// TIA Portal V17 export
// export: Created 2024-08-21T14:00:35.6590346Z, ExportSetting WithDefaults, DisplayName Totally Integrated Automation Portal, DisplayVersion V17 Update 4, DisplayName TIA Portal Openness, DisplayVersion V17 Update 4, DisplayName TIA Portal Version Control Interface, DisplayVersion V17, DisplayName STEP 7 Professional, DisplayVersion V17 Update 4, DisplayName STEP 7 Safety, DisplayVersion V17, DisplayName WinCC Advanced, DisplayVersion V17 Update 4
FUNCTION "IO" : Void   // FC1, LAD
{ S7_Optimized_Access := 'TRUE' }
VERSION : 0.1
// stored: AutoNumber false, IsIECCheckEnabled false, SetENOAutomatically false, UDAEnableTagReadback false
BEGIN

REGION Network 1: Status e alarme elevatória principal 1
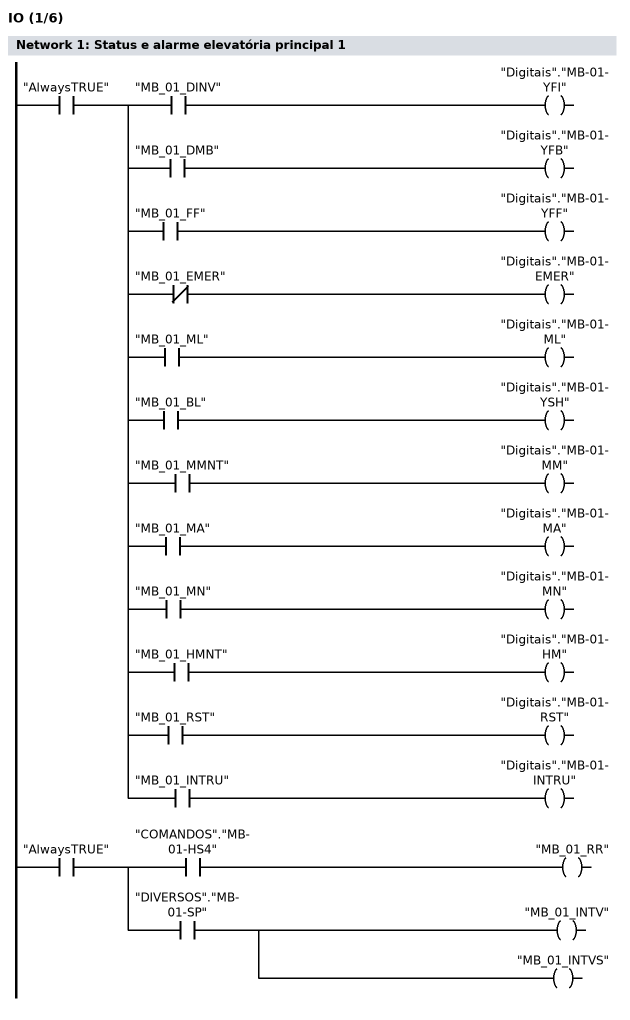
   RUNG wire#powerrail
      Contact( "AlwaysTRUE" )
      wire#w1
      Contact( "MB_01_DINV" )
      Coil( "Digitais"."MB-01-YFI" )
   END_RUNG
   RUNG wire#w1
      Contact( "MB_01_DMB" )
      Coil( "Digitais"."MB-01-YFB" )
   END_RUNG
   RUNG wire#w1
      Contact( "MB_01_FF" )
      Coil( "Digitais"."MB-01-YFF" )
   END_RUNG
   RUNG wire#w1
      I_Contact( "MB_01_EMER" )
      Coil( "Digitais"."MB-01-EMER" )
   END_RUNG
   RUNG wire#w1
      Contact( "MB_01_ML" )
      Coil( "Digitais"."MB-01-ML" )
   END_RUNG
   RUNG wire#w1
      Contact( "MB_01_BL" )
      Coil( "Digitais"."MB-01-YSH" )
   END_RUNG
   RUNG wire#w1
      Contact( "MB_01_MMNT" )
      Coil( "Digitais"."MB-01-MM" )
   END_RUNG
   RUNG wire#w1
      Contact( "MB_01_MA" )
      Coil( "Digitais"."MB-01-MA" )
   END_RUNG
   RUNG wire#w1
      Contact( "MB_01_MN" )
      Coil( "Digitais"."MB-01-MN" )
   END_RUNG
   RUNG wire#w1
      Contact( "MB_01_HMNT" )
      Coil( "Digitais"."MB-01-HM" )
   END_RUNG
   RUNG wire#w1
      Contact( "MB_01_RST" )
      Coil( "Digitais"."MB-01-RST" )
   END_RUNG
   RUNG wire#w1
      Contact( "MB_01_INTRU" )
      Coil( "Digitais"."MB-01-INTRU" )
   END_RUNG
   RUNG wire#powerrail
      Contact( "AlwaysTRUE" )
      wire#w2
      Contact( "COMANDOS"."MB-01-HS4" )
      Coil( "MB_01_RR" )
   END_RUNG
   RUNG wire#w2
      Contact( "DIVERSOS"."MB-01-SP" )
      wire#w3
      Coil( "MB_01_INTV" )
   END_RUNG
   RUNG wire#w3
      Coil( "MB_01_INTVS" )
   END_RUNG
   // the same network as SCL:
   "Digitais"."MB-01-YFI" := "AlwaysTRUE" AND "MB_01_DINV";
   "Digitais"."MB-01-YFB" := "AlwaysTRUE" AND "MB_01_DMB";
   "Digitais"."MB-01-YFF" := "AlwaysTRUE" AND "MB_01_FF";
   "Digitais"."MB-01-EMER" := "AlwaysTRUE" AND NOT "MB_01_EMER";
   "Digitais"."MB-01-ML" := "AlwaysTRUE" AND "MB_01_ML";
   "Digitais"."MB-01-YSH" := "AlwaysTRUE" AND "MB_01_BL";
   "Digitais"."MB-01-MM" := "AlwaysTRUE" AND "MB_01_MMNT";
   "Digitais"."MB-01-MA" := "AlwaysTRUE" AND "MB_01_MA";
   "Digitais"."MB-01-MN" := "AlwaysTRUE" AND "MB_01_MN";
   "Digitais"."MB-01-HM" := "AlwaysTRUE" AND "MB_01_HMNT";
   "Digitais"."MB-01-RST" := "AlwaysTRUE" AND "MB_01_RST";
   "Digitais"."MB-01-INTRU" := "AlwaysTRUE" AND "MB_01_INTRU";
   "MB_01_RR" := "AlwaysTRUE" AND "COMANDOS"."MB-01-HS4";
   "MB_01_INTV" := "AlwaysTRUE" AND "DIVERSOS"."MB-01-SP";
   "MB_01_INTVS" := "MB_01_INTV";
END_REGION

REGION Network 2: Status e alarme elevatória principal 2
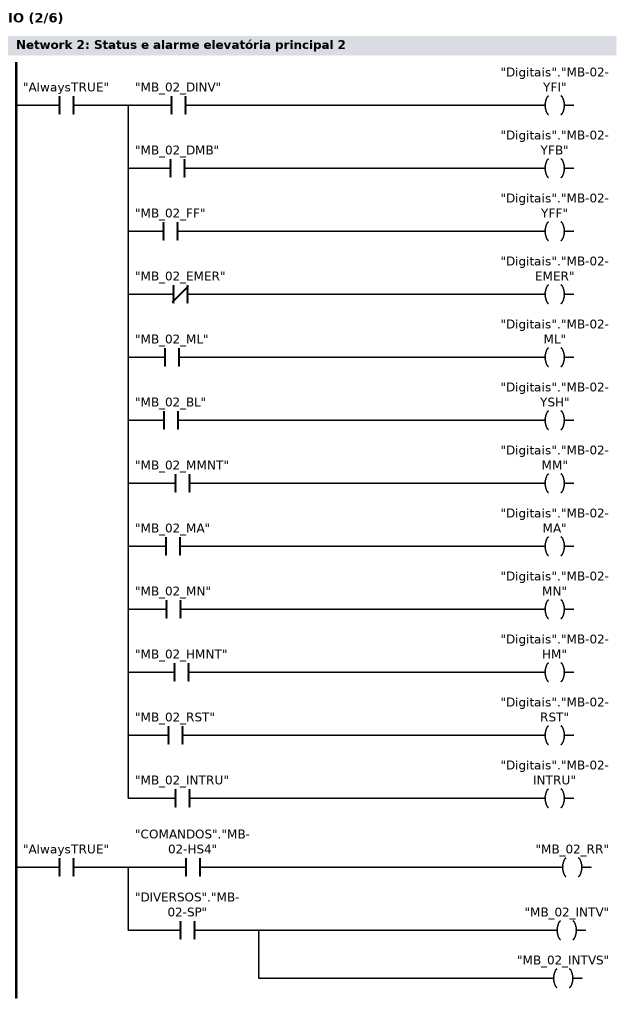
   RUNG wire#powerrail
      Contact( "AlwaysTRUE" )
      wire#w1
      Contact( "MB_02_DINV" )
      Coil( "Digitais"."MB-02-YFI" )
   END_RUNG
   RUNG wire#w1
      Contact( "MB_02_DMB" )
      Coil( "Digitais"."MB-02-YFB" )
   END_RUNG
   RUNG wire#w1
      Contact( "MB_02_FF" )
      Coil( "Digitais"."MB-02-YFF" )
   END_RUNG
   RUNG wire#w1
      I_Contact( "MB_02_EMER" )
      Coil( "Digitais"."MB-02-EMER" )
   END_RUNG
   RUNG wire#w1
      Contact( "MB_02_ML" )
      Coil( "Digitais"."MB-02-ML" )
   END_RUNG
   RUNG wire#w1
      Contact( "MB_02_BL" )
      Coil( "Digitais"."MB-02-YSH" )
   END_RUNG
   RUNG wire#w1
      Contact( "MB_02_MMNT" )
      Coil( "Digitais"."MB-02-MM" )
   END_RUNG
   RUNG wire#w1
      Contact( "MB_02_MA" )
      Coil( "Digitais"."MB-02-MA" )
   END_RUNG
   RUNG wire#w1
      Contact( "MB_02_MN" )
      Coil( "Digitais"."MB-02-MN" )
   END_RUNG
   RUNG wire#w1
      Contact( "MB_02_HMNT" )
      Coil( "Digitais"."MB-02-HM" )
   END_RUNG
   RUNG wire#w1
      Contact( "MB_02_RST" )
      Coil( "Digitais"."MB-02-RST" )
   END_RUNG
   RUNG wire#w1
      Contact( "MB_02_INTRU" )
      Coil( "Digitais"."MB-02-INTRU" )
   END_RUNG
   RUNG wire#powerrail
      Contact( "AlwaysTRUE" )
      wire#w2
      Contact( "COMANDOS"."MB-02-HS4" )
      Coil( "MB_02_RR" )
   END_RUNG
   RUNG wire#w2
      Contact( "DIVERSOS"."MB-02-SP" )
      wire#w3
      Coil( "MB_02_INTV" )
   END_RUNG
   RUNG wire#w3
      Coil( "MB_02_INTVS" )
   END_RUNG
   // the same network as SCL:
   "Digitais"."MB-02-YFI" := "AlwaysTRUE" AND "MB_02_DINV";
   "Digitais"."MB-02-YFB" := "AlwaysTRUE" AND "MB_02_DMB";
   "Digitais"."MB-02-YFF" := "AlwaysTRUE" AND "MB_02_FF";
   "Digitais"."MB-02-EMER" := "AlwaysTRUE" AND NOT "MB_02_EMER";
   "Digitais"."MB-02-ML" := "AlwaysTRUE" AND "MB_02_ML";
   "Digitais"."MB-02-YSH" := "AlwaysTRUE" AND "MB_02_BL";
   "Digitais"."MB-02-MM" := "AlwaysTRUE" AND "MB_02_MMNT";
   "Digitais"."MB-02-MA" := "AlwaysTRUE" AND "MB_02_MA";
   "Digitais"."MB-02-MN" := "AlwaysTRUE" AND "MB_02_MN";
   "Digitais"."MB-02-HM" := "AlwaysTRUE" AND "MB_02_HMNT";
   "Digitais"."MB-02-RST" := "AlwaysTRUE" AND "MB_02_RST";
   "Digitais"."MB-02-INTRU" := "AlwaysTRUE" AND "MB_02_INTRU";
   "MB_02_RR" := "AlwaysTRUE" AND "COMANDOS"."MB-02-HS4";
   "MB_02_INTV" := "AlwaysTRUE" AND "DIVERSOS"."MB-02-SP";
   "MB_02_INTVS" := "MB_02_INTV";
END_REGION

REGION Network 3: Status e alarme elevatória principal 3
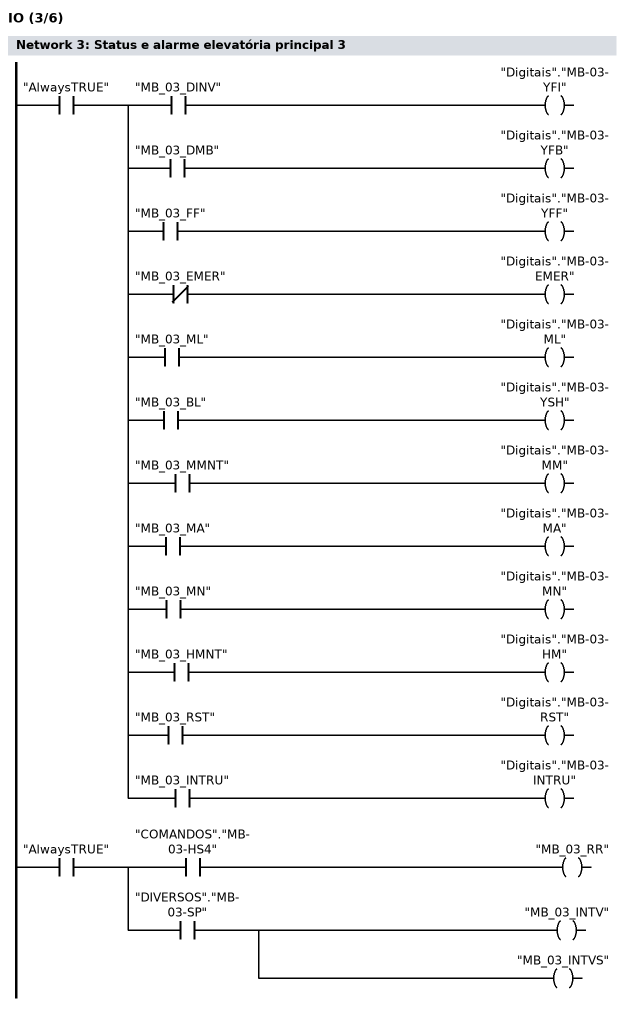
   RUNG wire#powerrail
      Contact( "AlwaysTRUE" )
      wire#w1
      Contact( "MB_03_DINV" )
      Coil( "Digitais"."MB-03-YFI" )
   END_RUNG
   RUNG wire#w1
      Contact( "MB_03_DMB" )
      Coil( "Digitais"."MB-03-YFB" )
   END_RUNG
   RUNG wire#w1
      Contact( "MB_03_FF" )
      Coil( "Digitais"."MB-03-YFF" )
   END_RUNG
   RUNG wire#w1
      I_Contact( "MB_03_EMER" )
      Coil( "Digitais"."MB-03-EMER" )
   END_RUNG
   RUNG wire#w1
      Contact( "MB_03_ML" )
      Coil( "Digitais"."MB-03-ML" )
   END_RUNG
   RUNG wire#w1
      Contact( "MB_03_BL" )
      Coil( "Digitais"."MB-03-YSH" )
   END_RUNG
   RUNG wire#w1
      Contact( "MB_03_MMNT" )
      Coil( "Digitais"."MB-03-MM" )
   END_RUNG
   RUNG wire#w1
      Contact( "MB_03_MA" )
      Coil( "Digitais"."MB-03-MA" )
   END_RUNG
   RUNG wire#w1
      Contact( "MB_03_MN" )
      Coil( "Digitais"."MB-03-MN" )
   END_RUNG
   RUNG wire#w1
      Contact( "MB_03_HMNT" )
      Coil( "Digitais"."MB-03-HM" )
   END_RUNG
   RUNG wire#w1
      Contact( "MB_03_RST" )
      Coil( "Digitais"."MB-03-RST" )
   END_RUNG
   RUNG wire#w1
      Contact( "MB_03_INTRU" )
      Coil( "Digitais"."MB-03-INTRU" )
   END_RUNG
   RUNG wire#powerrail
      Contact( "AlwaysTRUE" )
      wire#w2
      Contact( "COMANDOS"."MB-03-HS4" )
      Coil( "MB_03_RR" )
   END_RUNG
   RUNG wire#w2
      Contact( "DIVERSOS"."MB-03-SP" )
      wire#w3
      Coil( "MB_03_INTV" )
   END_RUNG
   RUNG wire#w3
      Coil( "MB_03_INTVS" )
   END_RUNG
   // the same network as SCL:
   "Digitais"."MB-03-YFI" := "AlwaysTRUE" AND "MB_03_DINV";
   "Digitais"."MB-03-YFB" := "AlwaysTRUE" AND "MB_03_DMB";
   "Digitais"."MB-03-YFF" := "AlwaysTRUE" AND "MB_03_FF";
   "Digitais"."MB-03-EMER" := "AlwaysTRUE" AND NOT "MB_03_EMER";
   "Digitais"."MB-03-ML" := "AlwaysTRUE" AND "MB_03_ML";
   "Digitais"."MB-03-YSH" := "AlwaysTRUE" AND "MB_03_BL";
   "Digitais"."MB-03-MM" := "AlwaysTRUE" AND "MB_03_MMNT";
   "Digitais"."MB-03-MA" := "AlwaysTRUE" AND "MB_03_MA";
   "Digitais"."MB-03-MN" := "AlwaysTRUE" AND "MB_03_MN";
   "Digitais"."MB-03-HM" := "AlwaysTRUE" AND "MB_03_HMNT";
   "Digitais"."MB-03-RST" := "AlwaysTRUE" AND "MB_03_RST";
   "Digitais"."MB-03-INTRU" := "AlwaysTRUE" AND "MB_03_INTRU";
   "MB_03_RR" := "AlwaysTRUE" AND "COMANDOS"."MB-03-HS4";
   "MB_03_INTV" := "AlwaysTRUE" AND "DIVERSOS"."MB-03-SP";
   "MB_03_INTVS" := "MB_03_INTV";
END_REGION

REGION Network 4: Status e alarme elevatória principal 4
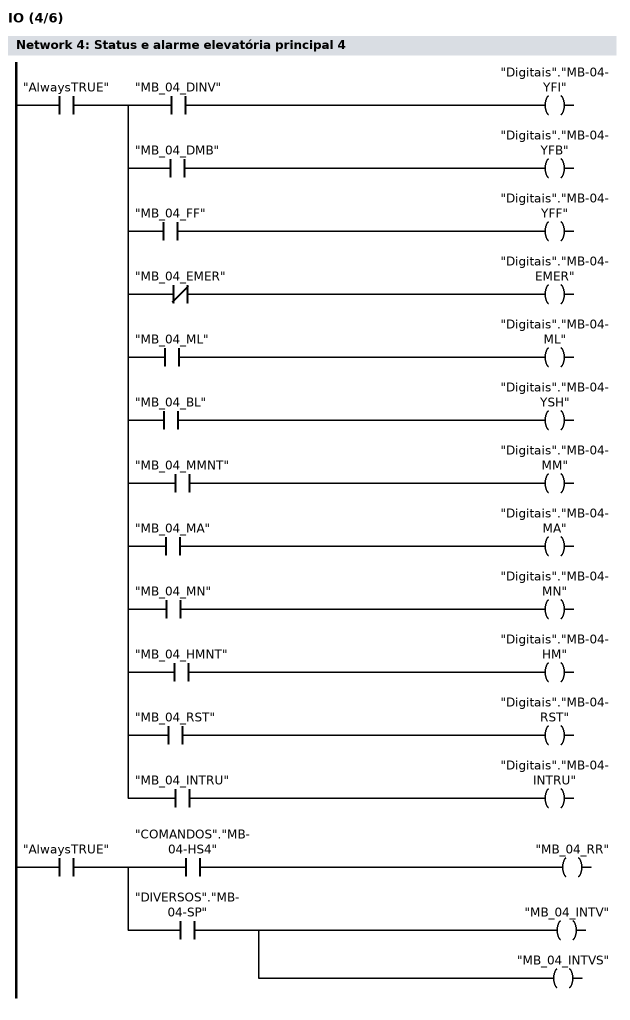
   RUNG wire#powerrail
      Contact( "AlwaysTRUE" )
      wire#w1
      Contact( "MB_04_DINV" )
      Coil( "Digitais"."MB-04-YFI" )
   END_RUNG
   RUNG wire#w1
      Contact( "MB_04_DMB" )
      Coil( "Digitais"."MB-04-YFB" )
   END_RUNG
   RUNG wire#w1
      Contact( "MB_04_FF" )
      Coil( "Digitais"."MB-04-YFF" )
   END_RUNG
   RUNG wire#w1
      I_Contact( "MB_04_EMER" )
      Coil( "Digitais"."MB-04-EMER" )
   END_RUNG
   RUNG wire#w1
      Contact( "MB_04_ML" )
      Coil( "Digitais"."MB-04-ML" )
   END_RUNG
   RUNG wire#w1
      Contact( "MB_04_BL" )
      Coil( "Digitais"."MB-04-YSH" )
   END_RUNG
   RUNG wire#w1
      Contact( "MB_04_MMNT" )
      Coil( "Digitais"."MB-04-MM" )
   END_RUNG
   RUNG wire#w1
      Contact( "MB_04_MA" )
      Coil( "Digitais"."MB-04-MA" )
   END_RUNG
   RUNG wire#w1
      Contact( "MB_04_MN" )
      Coil( "Digitais"."MB-04-MN" )
   END_RUNG
   RUNG wire#w1
      Contact( "MB_04_HMNT" )
      Coil( "Digitais"."MB-04-HM" )
   END_RUNG
   RUNG wire#w1
      Contact( "MB_04_RST" )
      Coil( "Digitais"."MB-04-RST" )
   END_RUNG
   RUNG wire#w1
      Contact( "MB_04_INTRU" )
      Coil( "Digitais"."MB-04-INTRU" )
   END_RUNG
   RUNG wire#powerrail
      Contact( "AlwaysTRUE" )
      wire#w2
      Contact( "COMANDOS"."MB-04-HS4" )
      Coil( "MB_04_RR" )
   END_RUNG
   RUNG wire#w2
      Contact( "DIVERSOS"."MB-04-SP" )
      wire#w3
      Coil( "MB_04_INTV" )
   END_RUNG
   RUNG wire#w3
      Coil( "MB_04_INTVS" )
   END_RUNG
   // the same network as SCL:
   "Digitais"."MB-04-YFI" := "AlwaysTRUE" AND "MB_04_DINV";
   "Digitais"."MB-04-YFB" := "AlwaysTRUE" AND "MB_04_DMB";
   "Digitais"."MB-04-YFF" := "AlwaysTRUE" AND "MB_04_FF";
   "Digitais"."MB-04-EMER" := "AlwaysTRUE" AND NOT "MB_04_EMER";
   "Digitais"."MB-04-ML" := "AlwaysTRUE" AND "MB_04_ML";
   "Digitais"."MB-04-YSH" := "AlwaysTRUE" AND "MB_04_BL";
   "Digitais"."MB-04-MM" := "AlwaysTRUE" AND "MB_04_MMNT";
   "Digitais"."MB-04-MA" := "AlwaysTRUE" AND "MB_04_MA";
   "Digitais"."MB-04-MN" := "AlwaysTRUE" AND "MB_04_MN";
   "Digitais"."MB-04-HM" := "AlwaysTRUE" AND "MB_04_HMNT";
   "Digitais"."MB-04-RST" := "AlwaysTRUE" AND "MB_04_RST";
   "Digitais"."MB-04-INTRU" := "AlwaysTRUE" AND "MB_04_INTRU";
   "MB_04_RR" := "AlwaysTRUE" AND "COMANDOS"."MB-04-HS4";
   "MB_04_INTV" := "AlwaysTRUE" AND "DIVERSOS"."MB-04-SP";
   "MB_04_INTVS" := "MB_04_INTV";
END_REGION

REGION Network 5: Status e alarme PCM-E-CF-01-04
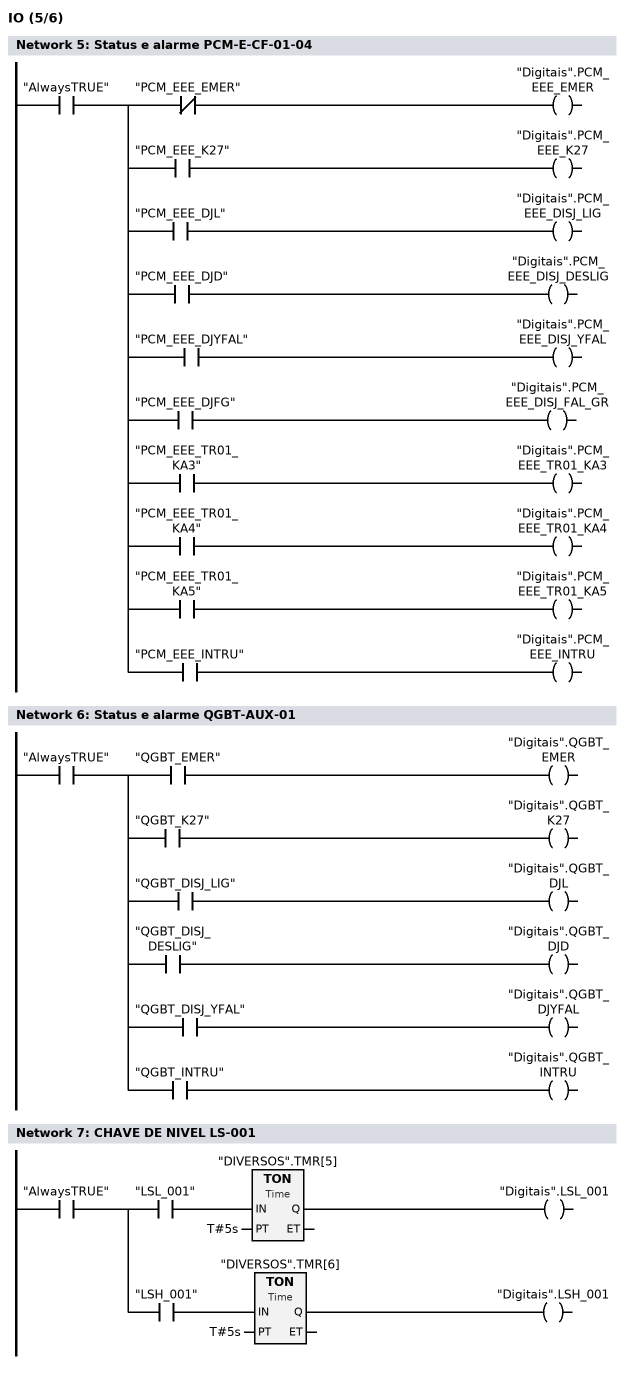
   RUNG wire#powerrail
      Contact( "AlwaysTRUE" )
      wire#w1
      I_Contact( "PCM_EEE_EMER" )
      Coil( "Digitais".PCM_EEE_EMER )
   END_RUNG
   RUNG wire#w1
      Contact( "PCM_EEE_K27" )
      Coil( "Digitais".PCM_EEE_K27 )
   END_RUNG
   RUNG wire#w1
      Contact( "PCM_EEE_DJL" )
      Coil( "Digitais".PCM_EEE_DISJ_LIG )
   END_RUNG
   RUNG wire#w1
      Contact( "PCM_EEE_DJD" )
      Coil( "Digitais".PCM_EEE_DISJ_DESLIG )
   END_RUNG
   RUNG wire#w1
      Contact( "PCM_EEE_DJYFAL" )
      Coil( "Digitais".PCM_EEE_DISJ_YFAL )
   END_RUNG
   RUNG wire#w1
      Contact( "PCM_EEE_DJFG" )
      Coil( "Digitais".PCM_EEE_DISJ_FAL_GR )
   END_RUNG
   RUNG wire#w1
      Contact( "PCM_EEE_TR01_KA3" )
      Coil( "Digitais".PCM_EEE_TR01_KA3 )
   END_RUNG
   RUNG wire#w1
      Contact( "PCM_EEE_TR01_KA4" )
      Coil( "Digitais".PCM_EEE_TR01_KA4 )
   END_RUNG
   RUNG wire#w1
      Contact( "PCM_EEE_TR01_KA5" )
      Coil( "Digitais".PCM_EEE_TR01_KA5 )
   END_RUNG
   RUNG wire#w1
      Contact( "PCM_EEE_INTRU" )
      Coil( "Digitais".PCM_EEE_INTRU )
   END_RUNG
   // the same network as SCL:
   "Digitais".PCM_EEE_EMER := "AlwaysTRUE" AND NOT "PCM_EEE_EMER";
   "Digitais".PCM_EEE_K27 := "AlwaysTRUE" AND "PCM_EEE_K27";
   "Digitais".PCM_EEE_DISJ_LIG := "AlwaysTRUE" AND "PCM_EEE_DJL";
   "Digitais".PCM_EEE_DISJ_DESLIG := "AlwaysTRUE" AND "PCM_EEE_DJD";
   "Digitais".PCM_EEE_DISJ_YFAL := "AlwaysTRUE" AND "PCM_EEE_DJYFAL";
   "Digitais".PCM_EEE_DISJ_FAL_GR := "AlwaysTRUE" AND "PCM_EEE_DJFG";
   "Digitais".PCM_EEE_TR01_KA3 := "AlwaysTRUE" AND "PCM_EEE_TR01_KA3";
   "Digitais".PCM_EEE_TR01_KA4 := "AlwaysTRUE" AND "PCM_EEE_TR01_KA4";
   "Digitais".PCM_EEE_TR01_KA5 := "AlwaysTRUE" AND "PCM_EEE_TR01_KA5";
   "Digitais".PCM_EEE_INTRU := "AlwaysTRUE" AND "PCM_EEE_INTRU";
END_REGION

REGION Network 6: Status e alarme QGBT-AUX-01
   RUNG wire#powerrail
      Contact( "AlwaysTRUE" )
      wire#w1
      Contact( "QGBT_EMER" )
      Coil( "Digitais".QGBT_EMER )
   END_RUNG
   RUNG wire#w1
      Contact( "QGBT_K27" )
      Coil( "Digitais".QGBT_K27 )
   END_RUNG
   RUNG wire#w1
      Contact( "QGBT_DISJ_LIG" )
      Coil( "Digitais".QGBT_DJL )
   END_RUNG
   RUNG wire#w1
      Contact( "QGBT_DISJ_DESLIG" )
      Coil( "Digitais".QGBT_DJD )
   END_RUNG
   RUNG wire#w1
      Contact( "QGBT_DISJ_YFAL" )
      Coil( "Digitais".QGBT_DJYFAL )
   END_RUNG
   RUNG wire#w1
      Contact( "QGBT_INTRU" )
      Coil( "Digitais".QGBT_INTRU )
   END_RUNG
   // the same network as SCL:
   "Digitais".QGBT_EMER := "AlwaysTRUE" AND "QGBT_EMER";
   "Digitais".QGBT_K27 := "AlwaysTRUE" AND "QGBT_K27";
   "Digitais".QGBT_DJL := "AlwaysTRUE" AND "QGBT_DISJ_LIG";
   "Digitais".QGBT_DJD := "AlwaysTRUE" AND "QGBT_DISJ_DESLIG";
   "Digitais".QGBT_DJYFAL := "AlwaysTRUE" AND "QGBT_DISJ_YFAL";
   "Digitais".QGBT_INTRU := "AlwaysTRUE" AND "QGBT_INTRU";
END_REGION

REGION Network 7: CHAVE DE NIVEL LS-001
   RUNG wire#powerrail
      Contact( "AlwaysTRUE" )
      wire#w1
      Contact( "LSL_001" )
      { S7_Templates := "time_type := Time" } "DIVERSOS".TMR[5].TON(pt := T#5s, et =>)
      Coil( "Digitais".LSL_001 )
   END_RUNG
   RUNG wire#w1
      Contact( "LSH_001" )
      { S7_Templates := "time_type := Time" } "DIVERSOS".TMR[6].TON(pt := T#5s, et =>)
      Coil( "Digitais".LSH_001 )
   END_RUNG
   // the same network as SCL:
   "DIVERSOS".TMR[5].TON(IN := "AlwaysTRUE" AND "LSL_001", PT := T#5s);
   "Digitais".LSL_001 := "DIVERSOS".TMR[5].Q;
   "DIVERSOS".TMR[6].TON(IN := "AlwaysTRUE" AND "LSH_001", PT := T#5s);
   "Digitais".LSH_001 := "DIVERSOS".TMR[6].Q;
END_REGION

REGION Network 8: CHAVE DE NIVEL LS-002
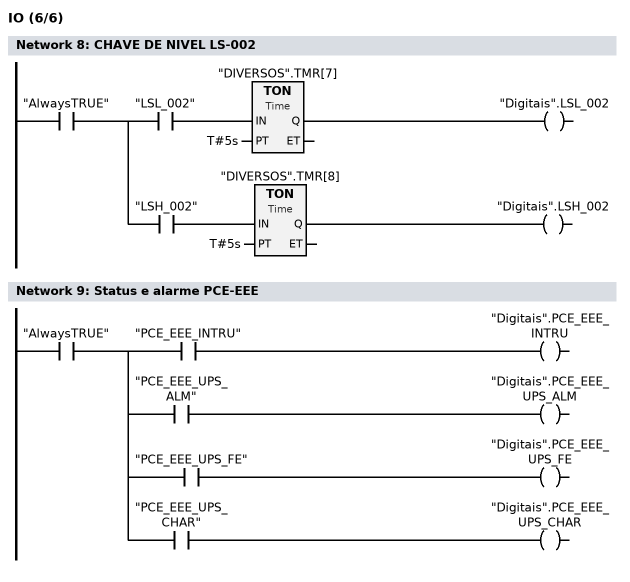
   RUNG wire#powerrail
      Contact( "AlwaysTRUE" )
      wire#w1
      Contact( "LSL_002" )
      { S7_Templates := "time_type := Time" } "DIVERSOS".TMR[7].TON(pt := T#5s, et =>)
      Coil( "Digitais".LSL_002 )
   END_RUNG
   RUNG wire#w1
      Contact( "LSH_002" )
      { S7_Templates := "time_type := Time" } "DIVERSOS".TMR[8].TON(pt := T#5s, et =>)
      Coil( "Digitais".LSH_002 )
   END_RUNG
   // the same network as SCL:
   "DIVERSOS".TMR[7].TON(IN := "AlwaysTRUE" AND "LSL_002", PT := T#5s);
   "Digitais".LSL_002 := "DIVERSOS".TMR[7].Q;
   "DIVERSOS".TMR[8].TON(IN := "AlwaysTRUE" AND "LSH_002", PT := T#5s);
   "Digitais".LSH_002 := "DIVERSOS".TMR[8].Q;
END_REGION

REGION Network 9: Status e alarme PCE-EEE
   RUNG wire#powerrail
      Contact( "AlwaysTRUE" )
      wire#w1
      Contact( "PCE_EEE_INTRU" )
      Coil( "Digitais".PCE_EEE_INTRU )
   END_RUNG
   RUNG wire#w1
      Contact( "PCE_EEE_UPS_ALM" )
      Coil( "Digitais".PCE_EEE_UPS_ALM )
   END_RUNG
   RUNG wire#w1
      Contact( "PCE_EEE_UPS_FE" )
      Coil( "Digitais".PCE_EEE_UPS_FE )
   END_RUNG
   RUNG wire#w1
      Contact( "PCE_EEE_UPS_CHAR" )
      Coil( "Digitais".PCE_EEE_UPS_CHAR )
   END_RUNG
   // the same network as SCL:
   "Digitais".PCE_EEE_INTRU := "AlwaysTRUE" AND "PCE_EEE_INTRU";
   "Digitais".PCE_EEE_UPS_ALM := "AlwaysTRUE" AND "PCE_EEE_UPS_ALM";
   "Digitais".PCE_EEE_UPS_FE := "AlwaysTRUE" AND "PCE_EEE_UPS_FE";
   "Digitais".PCE_EEE_UPS_CHAR := "AlwaysTRUE" AND "PCE_EEE_UPS_CHAR";
END_REGION
END_FUNCTION
